(* PLC project ammonium-nitrates, Generated TextualNotationConverter 1.0 *)
(* stored: creationDateTime 2025-07-30T12:00:00, modificationDateTime 2025-09-27T11:37:37 *)

FUNCTION_BLOCK ANALOG_IN
  VAR_INPUT
    Name : STRING;
    Description : STRING;
    Raw_Signal : REAL;
    PV_High : REAL;
    PV_Low : REAL;
    Scaling_Slope : REAL;
    Scaling_Offset : REAL;
    Alarm_Enable : BOOL;
  END_VAR
  VAR_OUTPUT
    PV : REAL;
    High_Alarm : BOOL;
    Low_Alarm : BOOL;
    General_Fault : BOOL;
  END_VAR

            
          
END_FUNCTION_BLOCK

FUNCTION_BLOCK BOOL_IN
  VAR_INPUT
    Name : STRING;
    Description : STRING;
    Bool_In : BOOL;
    Alarm_OnTrue : BOOL;
    Alarm_OnFalse : BOOL;
    Latch_Enable : BOOL;
    Reset_Latch : BOOL;
  END_VAR
  VAR_OUTPUT
    Bool_Out : BOOL;
    Alarm_Active : BOOL;
    Latched_Status : BOOL;
  END_VAR

            
          
END_FUNCTION_BLOCK

FUNCTION_BLOCK PID_BASIC
  VAR_INPUT
    Name : STRING;
    Description : STRING;
    AUTO : BOOL;
    PV : REAL;
    SP : REAL;
    MV_MIN : REAL;
    MV_MAX : REAL;
    X0 : REAL;
    KP : REAL;
    TR : REAL;
    TD : REAL;
    PV_High : REAL;
    PV_Low : REAL;
    Deviation_Limit : REAL;
    Inhibit : BOOL;
  END_VAR
  VAR_OUTPUT
    PV_High_Alarm : BOOL;
    PV_Low_Alarm : BOOL;
    Deviation_Alarm : BOOL;
    XOUT : REAL;
  END_VAR

            
          
END_FUNCTION_BLOCK

FUNCTION_BLOCK RATIO_CONTROL
  VAR_INPUT
    Name : STRING;
    Description : STRING;
    Auto : BOOL;
    PrimaryPV : REAL;
    SecondaryPV : REAL;
    RatioSP : REAL;
    Bias : REAL;
    TrimKp : REAL;
    TrimTi : STRING;
    MV_MIN : REAL;
    MV_MAX : REAL;
    ManOut : REAL;
    Inhibit : BOOL;
  END_VAR
  VAR_OUTPUT
    SlaveSP : REAL;
    ActiveRatio : REAL;
    RatioErr : REAL;
  END_VAR

            
          
END_FUNCTION_BLOCK

FUNCTION_BLOCK VALVE_ELECTRIC
  VAR_INPUT
    Name : STRING;
    Description : STRING;
    Control_Signal : REAL;
    Manual_Mode : BOOL;
    Manual_Position : REAL;
    Open_Limit : REAL;
    Close_Limit : REAL;
    Timeout : STRING;
    Inhibit : BOOL;
  END_VAR
  VAR_OUTPUT
    Valve_Position : REAL;
    Feedback_Pos : REAL;
    Valve_Moving : BOOL;
    Position_Error : BOOL;
    Alarm : BOOL;
  END_VAR

            
          
END_FUNCTION_BLOCK

PROGRAM Section2
  VAR
    FIC102_AcidFlow_SP_FromRatio : REAL;
    FT101_AmmoniaFlow_PV : REAL;
    LT104_ReactorLevel_PV : REAL;
    PH105_ReactorPH_PV : REAL;
    VS107_Scrubber_Permissive : BOOL;
    VS107_Scrubber_Running_DI : BOOL;
    FT101_Raw_mA : REAL;
    FT102_Raw_mA : REAL;
    LT104_Raw_mA : REAL;
    PH105_Raw_mA : REAL;
    TIC103_Temperature_PV : REAL;
  END_VAR
  VAR
    FFIC-102 : RATIO_CONTROL;
    FIC-102 : PID_BASIC;
    FIC-101 : PID_BASIC;
    TIC-103 : PID_BASIC;
    FT-101 : ANALOG_IN;
    FT-102 : ANALOG_IN;
    LT-104 : ANALOG_IN;
    PH-105 : ANALOG_IN;
    FV-102 : VALVE_ELECTRIC;
    FV-101 : VALVE_ELECTRIC;
    VS-107 : BOOL_IN;
  END_VAR
  VAR  (* added by the conversion: wires and edge detectors of the diagram *)
    _OR1_OUT : BOOL;
    _OR3_OUT : BOOL;
  END_VAR

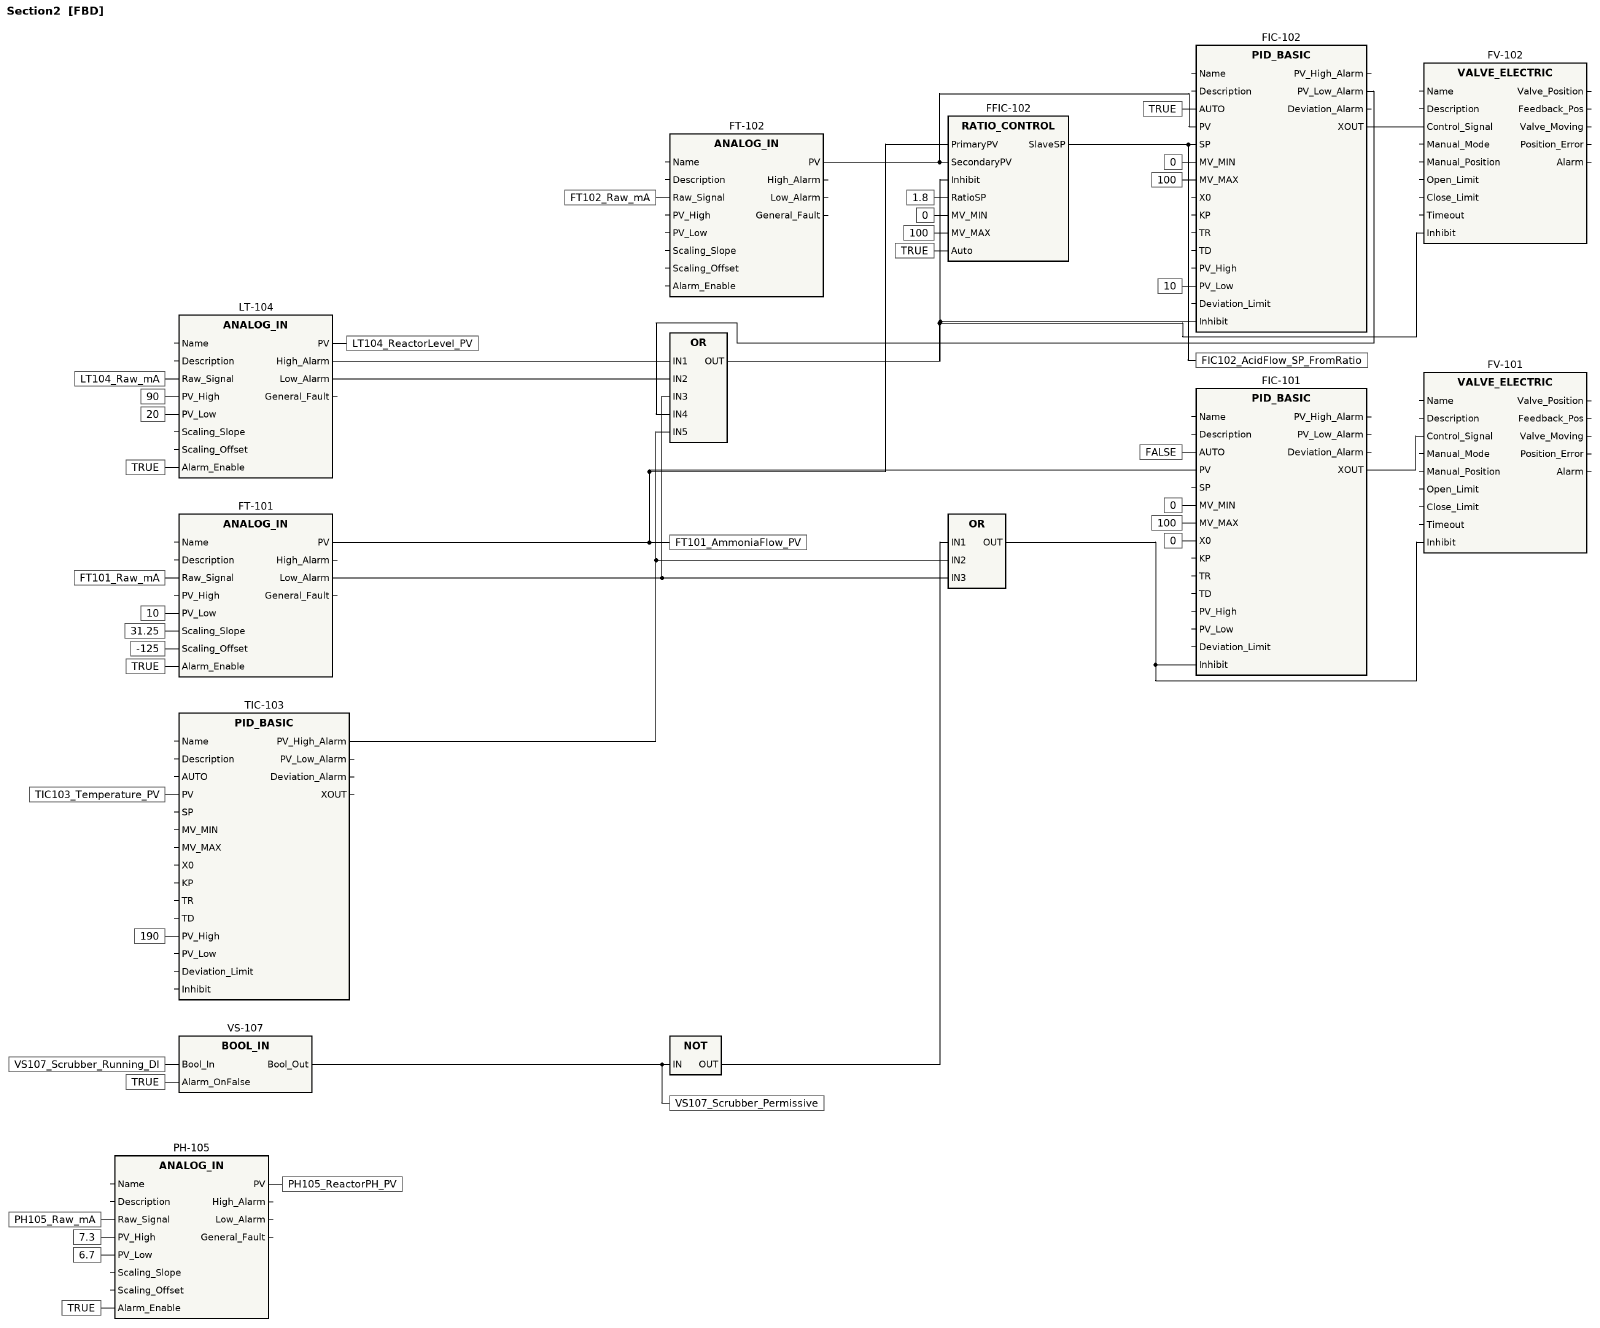
(* FBD diagram, written out as Structured Text *)
FT-101(Raw_Signal := FT101_Raw_mA, PV_Low := 10, Scaling_Slope := 31.25, Scaling_Offset := -125, Alarm_Enable := TRUE);
FT-102(Raw_Signal := FT102_Raw_mA);
LT-104(Raw_Signal := LT104_Raw_mA, PV_High := 90, PV_Low := 20, Alarm_Enable := TRUE);
FIC-102(AUTO := TRUE, PV := FT-102.PV, SP := FFIC-102.SlaveSP, MV_MIN := 0, MV_MAX := 100, PV_Low := 10, Inhibit := _OR1_OUT);
TIC-103(PV := TIC103_Temperature_PV, PV_High := 190);
_OR1_OUT := LT-104.High_Alarm OR LT-104.Low_Alarm OR FT-101.Low_Alarm OR FIC-102.PV_Low_Alarm OR TIC-103.PV_High_Alarm;
FFIC-102(PrimaryPV := FT-101.PV, SecondaryPV := FT-102.PV, Inhibit := _OR1_OUT, RatioSP := 1.8, MV_MIN := 0, MV_MAX := 100, Auto := TRUE);
FIC102_AcidFlow_SP_FromRatio := FFIC-102.SlaveSP;
FT101_AmmoniaFlow_PV := FT-101.PV;
LT104_ReactorLevel_PV := LT-104.PV;
PH-105(Raw_Signal := PH105_Raw_mA, PV_High := 7.3, PV_Low := 6.7, Alarm_Enable := TRUE);
PH105_ReactorPH_PV := PH-105.PV;
VS-107(Bool_In := VS107_Scrubber_Running_DI, Alarm_OnFalse := TRUE);
VS107_Scrubber_Permissive := VS-107.Bool_Out;
_OR3_OUT := NOT VS-107.Bool_Out OR TIC-103.PV_High_Alarm OR FT-101.Low_Alarm;
FIC-101(AUTO := FALSE, PV := FT-101.PV, MV_MIN := 0, MV_MAX := 100, X0 := 0, Inhibit := _OR3_OUT);
FV-102(Control_Signal := FIC-102.XOUT, Inhibit := _OR1_OUT);
FV-101(Control_Signal := FIC-101.XOUT, Inhibit := _OR3_OUT);
END_PROGRAM

FUNCTION_BLOCK DIGITAL_IN
  VAR_INPUT
    Name : STRING;
    Description : STRING;
    DI_Raw : BOOL;
    DebounceTime : STRING;
    EnableAlarm : BOOL;
  END_VAR
  VAR_OUTPUT
    DI_Out : BOOL;
    Fault_State : BOOL;
  END_VAR

            
          
END_FUNCTION_BLOCK

FUNCTION_BLOCK DUTY_STANDBY
  VAR_INPUT
    Name : STRING;
    Description : STRING;
    Enable : BOOL;
    StartRequest : BOOL;
    AlternateEnable : BOOL;
    ForcePumpA : BOOL;
    ForcePumpB : BOOL;
    DutyElapsed : BOOL;
    MinRunElapsed : BOOL;
    SwitchoverDelayElapsed : BOOL;
    StartTimeoutElapsed : BOOL;
    PumpA_RunFB : BOOL;
    PumpB_RunFB : BOOL;
    PumpA_Fault : BOOL;
    PumpB_Fault : BOOL;
    Reset : BOOL;
    Inhibit : BOOL;
  END_VAR
  VAR_OUTPUT
    CmdPumpA : BOOL;
    CmdPumpB : BOOL;
    ActiveIsA : BOOL;
    SwitchedDueToDuty : BOOL;
    SwitchedDueToFailure : BOOL;
    Alarm_FailedStart_A : BOOL;
    Alarm_FailedStart_B : BOOL;
    Alarm_NoAvailablePump : BOOL;
  END_VAR

            
          
END_FUNCTION_BLOCK

FUNCTION_BLOCK MOTOR_2SPD
  VAR_INPUT
    Name : STRING;
    Description : STRING;
    Start_Cmd : BOOL;
    Stop_Cmd : BOOL;
    Speed_High_Cmd : BOOL;
    Speed_Low_Cmd : BOOL;
    Inhibit : BOOL;
  END_VAR
  VAR_OUTPUT
    Motor_Start_Out : BOOL;
    FB_Running : BOOL;
    FB_Trip : BOOL;
    FB_HighSpeed : BOOL;
    FB_LowSpeed : BOOL;
    Alarm_Speed_Error : BOOL;
  END_VAR

            
          
END_FUNCTION_BLOCK

FUNCTION_BLOCK MOTOR_ON_OFF
  VAR_INPUT
    Name : STRING;
    Description : STRING;
    Start_Cmd : BOOL;
    Stop_Cmd : BOOL;
    Start_Delay : STRING;
    MinRunTime : STRING;
    Inhibit : BOOL;
  END_VAR
  VAR_OUTPUT
    Motor_Start_Out : BOOL;
    FB_Running : BOOL;
    FB_Trip : BOOL;
    Alarm_Start_Fail : BOOL;
    Alarm_Stop_Fail : BOOL;
  END_VAR

            
          
END_FUNCTION_BLOCK

FUNCTION_BLOCK MOTOR_VSD
  VAR_INPUT
    Name : STRING;
    Description : STRING;
    Start_Cmd : BOOL;
    Stop_Cmd : BOOL;
    Speed_SP : REAL;
    Accel_Ramp : STRING;
    Decel_Ramp : STRING;
    Inhibit : BOOL;
  END_VAR
  VAR_OUTPUT
    Speed_Out : REAL;
    FB_Running : BOOL;
    FB_Fault : BOOL;
    FB_Ready : BOOL;
    FB_ActualSpeed : REAL;
    Alarm_Speed_Deviation : BOOL;
    Alarm_Comm_Fail : BOOL;
  END_VAR

            
          
END_FUNCTION_BLOCK

FUNCTION_BLOCK SPLIT_RANGE
  VAR_INPUT
    Name : STRING;
    Description : STRING;
    IN : REAL;
    Split_Point : REAL;
    Output1_Start : REAL;
    Output1_End : REAL;
    Output2_Start : REAL;
    Output2_End : REAL;
  END_VAR
  VAR_OUTPUT
    OUT1 : REAL;
    OUT2 : REAL;
  END_VAR

            
          
END_FUNCTION_BLOCK

FUNCTION_BLOCK VALVE_ON_OFF
  VAR_INPUT
    Name : STRING;
    Description : STRING;
    Open_Cmd : BOOL;
    Close_Cmd : BOOL;
    Timeout : STRING;
    Inhibit : BOOL;
  END_VAR
  VAR_OUTPUT
    FB_Opened : BOOL;
    FB_Closed : BOOL;
    Valve_Open_Out : BOOL;
    Valve_Close_Out : BOOL;
    Alarm_Position_Error : BOOL;
    Alarm_General : BOOL;
  END_VAR

            
          
END_FUNCTION_BLOCK

FUNCTION_BLOCK VOTING_ANALOG
  VAR_INPUT
    Name : STRING;
    Description : STRING;
    Input1 : REAL;
    Input2 : REAL;
    Input3 : REAL;
    Deviation_Limit : REAL;
    Voting_Scheme : STRING;
    EnableAlarm : BOOL;
    Inhibit : BOOL;
  END_VAR
  VAR_OUTPUT
    Voted_Output : REAL;
    Sensor1_Fault : BOOL;
    Sensor2_Fault : BOOL;
    Sensor3_Fault : BOOL;
    Alarm_Voting_Error : BOOL;
    Healthy_Sensors_Count : INT;
  END_VAR

            
          
END_FUNCTION_BLOCK

PROGRAM Section3
  VAR
    TIC201_RSP_to_FIC102 : REAL;
  END_VAR
  VAR
    TT-103 : ANALOG_IN;
    TT-104 : ANALOG_IN;
    PT-203 : ANALOG_IN;
    TIC-201 : PID_BASIC;
    FIC-102 : PID_BASIC;
    FV-102 : VALVE_ELECTRIC;
    PV-106 : VALVE_ELECTRIC;
    XV-101 : VALVE_ON_OFF;
    P-205 : MOTOR_ON_OFF;
    HS-204 : DIGITAL_IN;
    VS-206 : DIGITAL_IN;
  END_VAR
  VAR  (* added by the conversion: wires and edge detectors of the diagram *)
    _OR281_OUT : BOOL;
    _OR282_OUT : BOOL;
    _OR283_OUT : BOOL;
  END_VAR

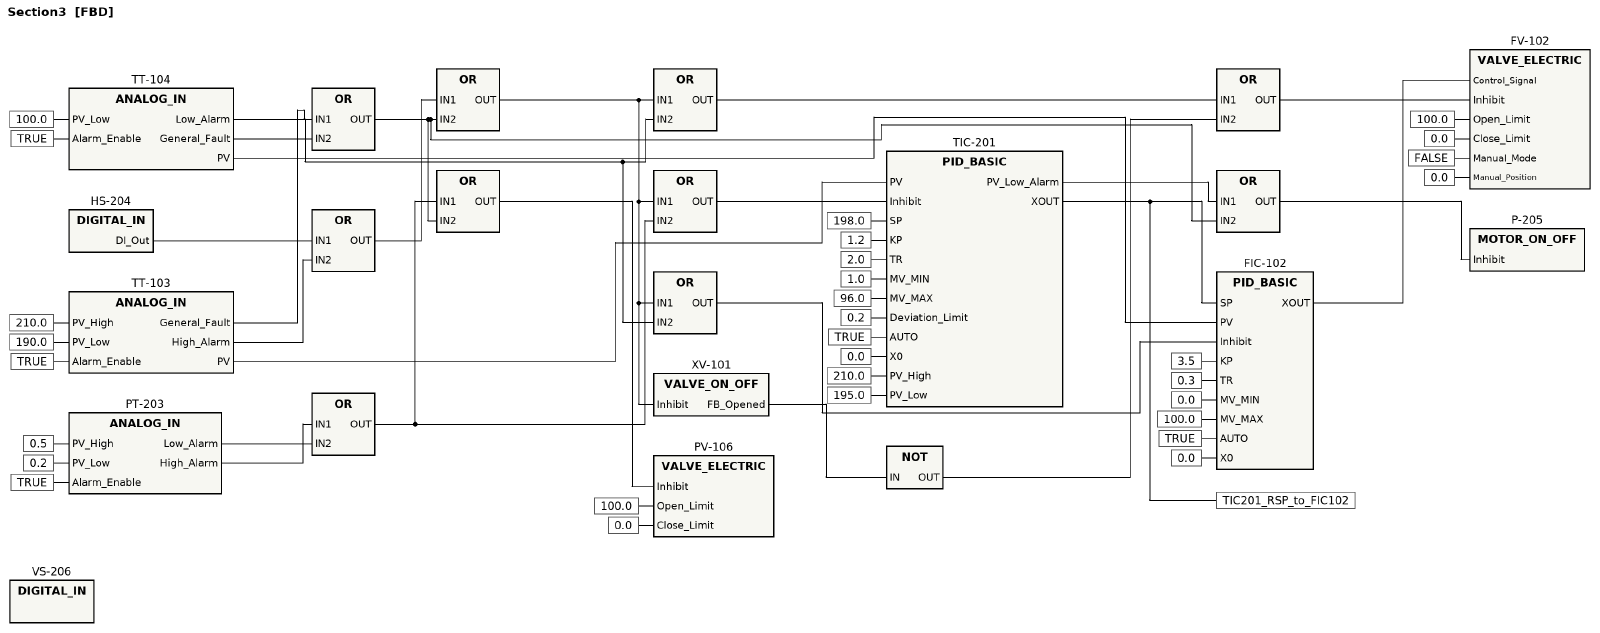
(* FBD diagram, written out as Structured Text *)
TT-103(PV_High := 210.0, PV_Low := 190.0, Alarm_Enable := TRUE);
HS-204();
TT-104(PV_Low := 100.0, Alarm_Enable := TRUE);
_OR281_OUT := TT-103.General_Fault OR TT-104.General_Fault;
_OR282_OUT := HS-204.DI_Out OR TT-103.High_Alarm OR _OR281_OUT;
PT-203(PV_High := 0.5, PV_Low := 0.2, Alarm_Enable := TRUE);
_OR283_OUT := PT-203.High_Alarm OR PT-203.Low_Alarm;
TIC-201(PV := TT-103.PV, Inhibit := _OR282_OUT OR _OR283_OUT, SP := 198.0, KP := 1.2, TR := 2.0, MV_MIN := 1.0, MV_MAX := 96.0, Deviation_Limit := 0.2, AUTO := TRUE, X0 := 0.0, PV_High := 210.0, PV_Low := 195.0);
TIC201_RSP_to_FIC102 := TIC-201.XOUT;
XV-101(Inhibit := _OR282_OUT);
FIC-102(SP := TIC-201.XOUT, PV := TT-104.PV, Inhibit := _OR282_OUT OR TT-104.Low_Alarm, KP := 3.5, TR := 0.3, MV_MIN := 0.0, MV_MAX := 100.0, AUTO := TRUE, X0 := 0.0);
FV-102(Control_Signal := FIC-102.XOUT, Inhibit := _OR282_OUT OR TT-104.Low_Alarm OR NOT XV-101.FB_Opened, Open_Limit := 100.0, Close_Limit := 0.0, Manual_Mode := FALSE, Manual_Position := 0.0);
PV-106(Inhibit := _OR283_OUT OR _OR281_OUT, Open_Limit := 100.0, Close_Limit := 0.0);
P-205(Inhibit := TIC-201.PV_Low_Alarm OR _OR281_OUT);
VS-206();
END_PROGRAM

PROGRAM Section4
  VAR
    RTD302_BedTemp_PV : REAL;
    FT301_Flow_PV : REAL;
    TIC302_RSP_to_FIC301 : REAL;
    FIC301_MV_Out_to_FV301 : REAL;
    AT303_Humidity_PV : REAL;
    PR305_TowerPressure_PV : REAL;
    VS304_Vibration_PV : REAL;
  END_VAR
  VAR
    AT-303 : ANALOG_IN;
    FIC-301 : PID_BASIC;
    FT-301 : ANALOG_IN;
    FV-301 : VALVE_ELECTRIC;
    PR-305 : ANALOG_IN;
    RTD-302 : ANALOG_IN;
    TIC-302 : PID_BASIC;
    VS-304 : ANALOG_IN;
    GR-306 : BOOL_IN;
  END_VAR

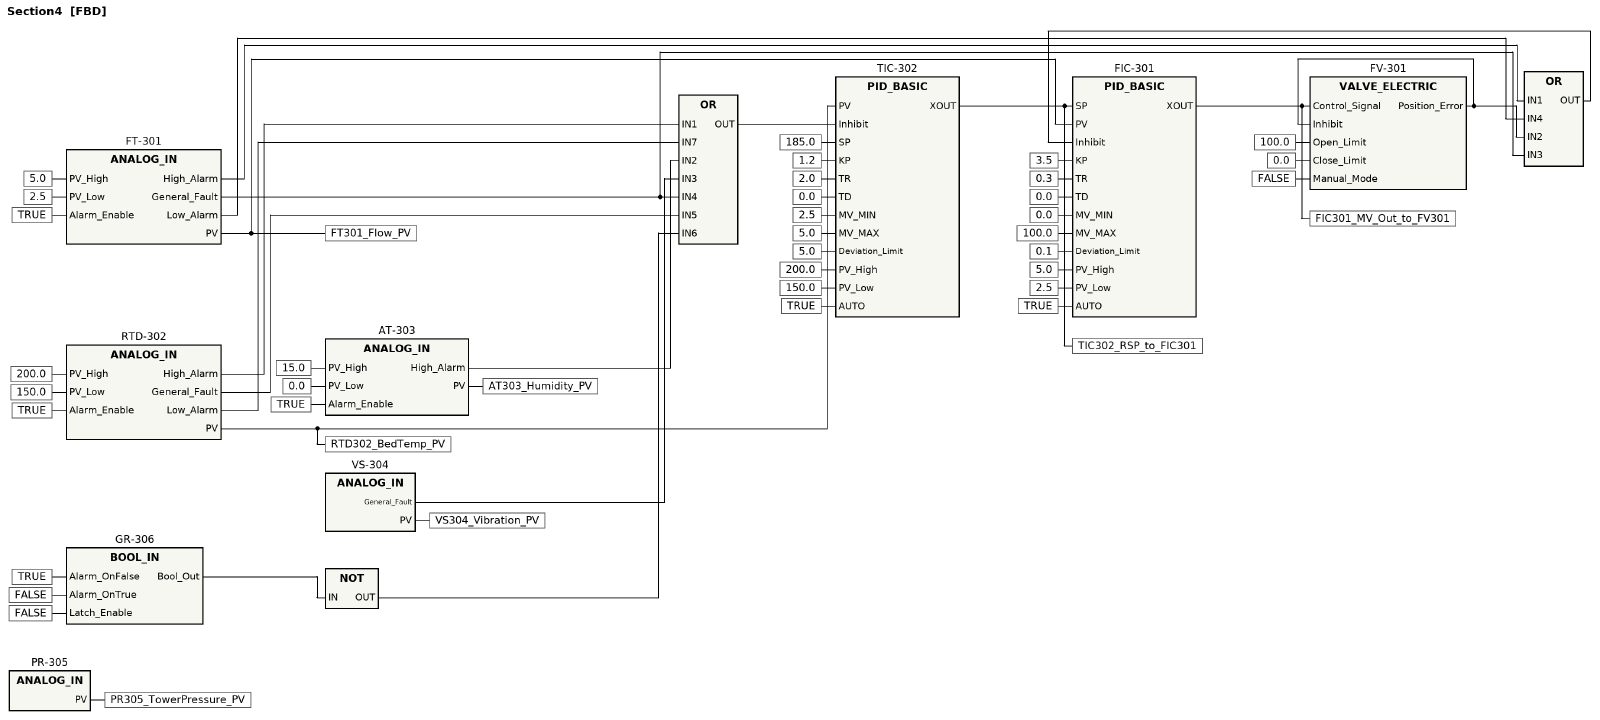
(* FBD diagram, written out as Structured Text *)
AT-303(PV_High := 15.0, PV_Low := 0.0, Alarm_Enable := TRUE);
AT303_Humidity_PV := AT-303.PV;
RTD-302(PV_High := 200.0, PV_Low := 150.0, Alarm_Enable := TRUE);
VS-304();
FT-301(PV_High := 5.0, PV_Low := 2.5, Alarm_Enable := TRUE);
GR-306(Alarm_OnFalse := TRUE, Alarm_OnTrue := FALSE, Latch_Enable := FALSE);
TIC-302(PV := RTD-302.PV, Inhibit := RTD-302.High_Alarm OR RTD-302.Low_Alarm OR AT-303.High_Alarm OR VS-304.General_Fault OR FT-301.General_Fault OR RTD-302.General_Fault OR NOT GR-306.Bool_Out, SP := 185.0, KP := 1.2, TR := 2.0, TD := 0.0, MV_MIN := 2.5, MV_MAX := 5.0, Deviation_Limit := 5.0, PV_High := 200.0, PV_Low := 150.0, AUTO := TRUE);
FV-301(Control_Signal := FIC-301.XOUT, Inhibit := FV-301.Position_Error, Open_Limit := 100.0, Close_Limit := 0.0, Manual_Mode := FALSE);
FIC-301(SP := TIC-302.XOUT, PV := FT-301.PV, Inhibit := FT-301.High_Alarm OR FT-301.Low_Alarm OR FV-301.Position_Error OR FT-301.General_Fault, KP := 3.5, TR := 0.3, TD := 0.0, MV_MIN := 0.0, MV_MAX := 100.0, Deviation_Limit := 0.1, PV_High := 5.0, PV_Low := 2.5, AUTO := TRUE);
FIC301_MV_Out_to_FV301 := FIC-301.XOUT;
FT301_Flow_PV := FT-301.PV;
PR-305();
PR305_TowerPressure_PV := PR-305.PV;
RTD302_BedTemp_PV := RTD-302.PV;
TIC302_RSP_to_FIC301 := TIC-302.XOUT;
VS304_Vibration_PV := VS-304.PV;
END_PROGRAM

PROGRAM Section5
  VAR
    TT401_CoolerOutletTemp_PV : REAL;
    FT402_AntiCakingFlow_PV : REAL;
    TIC401_RSP_to_FIC402 : REAL;
    FIC402_MV_to_FV402 : REAL;
    FIC402_SP_Manual : REAL;
  END_VAR
  VAR
    TIC-401 : PID_BASIC;
    TT-401 : ANALOG_IN;
    FIC-402 : PID_BASIC;
    FT-402 : ANALOG_IN;
    FV-402 : VALVE_ELECTRIC;
    MP-405 : MOTOR_ON_OFF;
    PS-403 : BOOL_IN;
    PSA-404 : DIGITAL_IN;
  END_VAR
  VAR  (* added by the conversion: wires and edge detectors of the diagram *)
    _OR184_OUT : BOOL;
  END_VAR

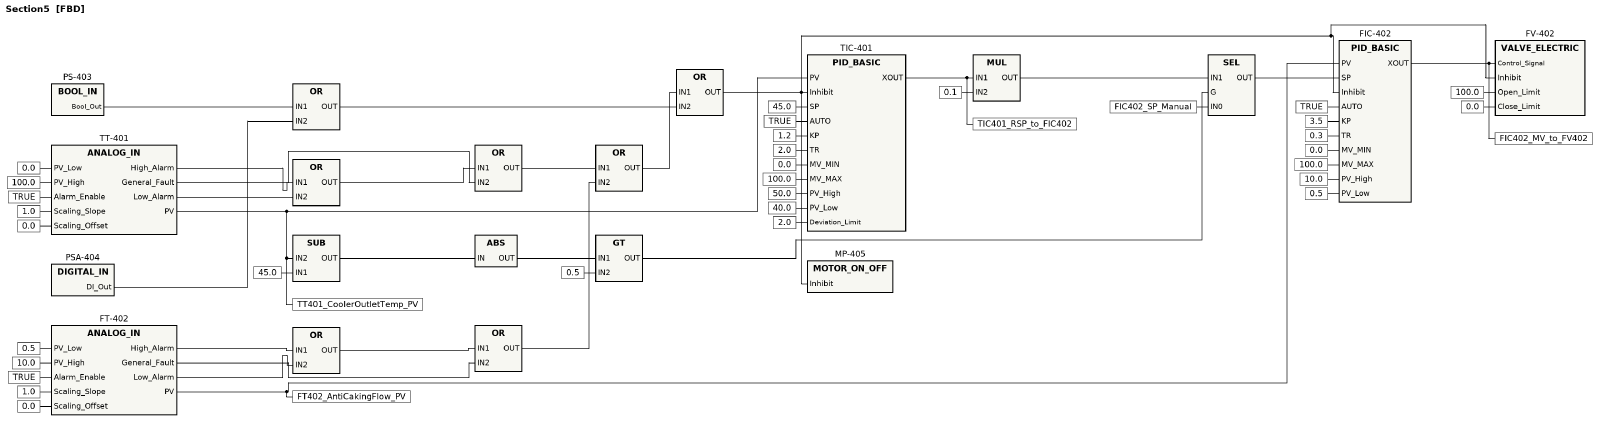
(* FBD diagram, written out as Structured Text *)
FT-402(PV_Low := 0.5, PV_High := 10.0, Alarm_Enable := TRUE, Scaling_Slope := 1.0, Scaling_Offset := 0.0);
TT-401(PV_Low := 0.0, PV_High := 100.0, Alarm_Enable := TRUE, Scaling_Slope := 1.0, Scaling_Offset := 0.0);
PS-403();
PSA-404();
_OR184_OUT := TT-401.High_Alarm OR TT-401.Low_Alarm OR TT-401.General_Fault OR FT-402.High_Alarm OR FT-402.Low_Alarm OR FT-402.General_Fault OR PS-403.Bool_Out OR PSA-404.DI_Out;
TIC-401(PV := TT-401.PV, Inhibit := _OR184_OUT, SP := 45.0, AUTO := TRUE, KP := 1.2, TR := 2.0, MV_MIN := 0.0, MV_MAX := 100.0, PV_High := 50.0, PV_Low := 40.0, Deviation_Limit := 2.0);
FIC-402(PV := FT-402.PV, SP := SEL(TIC-401.XOUT * 0.1, ABS(TT-401.PV - 45.0) > 0.5, FIC402_SP_Manual), Inhibit := _OR184_OUT, AUTO := TRUE, KP := 3.5, TR := 0.3, MV_MIN := 0.0, MV_MAX := 100.0, PV_High := 10.0, PV_Low := 0.5);
FIC402_MV_to_FV402 := FIC-402.XOUT;
FT402_AntiCakingFlow_PV := FT-402.PV;
TIC401_RSP_to_FIC402 := TIC-401.XOUT;
TT401_CoolerOutletTemp_PV := TT-401.PV;
FV-402(Control_Signal := FIC-402.XOUT, Inhibit := _OR184_OUT, Open_Limit := 100.0, Close_Limit := 0.0);
MP-405(Inhibit := _OR184_OUT);
END_PROGRAM

PROGRAM Section6
  VAR
    LT501_Level_Pct : REAL;
    WB505_Flow_Pct : REAL;
    RIC506_SC504_FlowSP : REAL;
    Ratio_Bias_Manual : REAL;
  END_VAR
  VAR
    LT-501 : ANALOG_IN;
    WB-505 : ANALOG_IN;
    AP-503 : VALVE_ON_OFF;
    PRV-502 : VALVE_ON_OFF;
    RIC-506 : RATIO_CONTROL;
    FIC-507 : PID_BASIC;
    SC-504 : MOTOR_VSD;
  END_VAR
  VAR  (* added by the conversion: wires and edge detectors of the diagram *)
    _OR232_OUT : BOOL;
    _GT233_OUT : BOOL;
    _LT234_OUT : BOOL;
  END_VAR

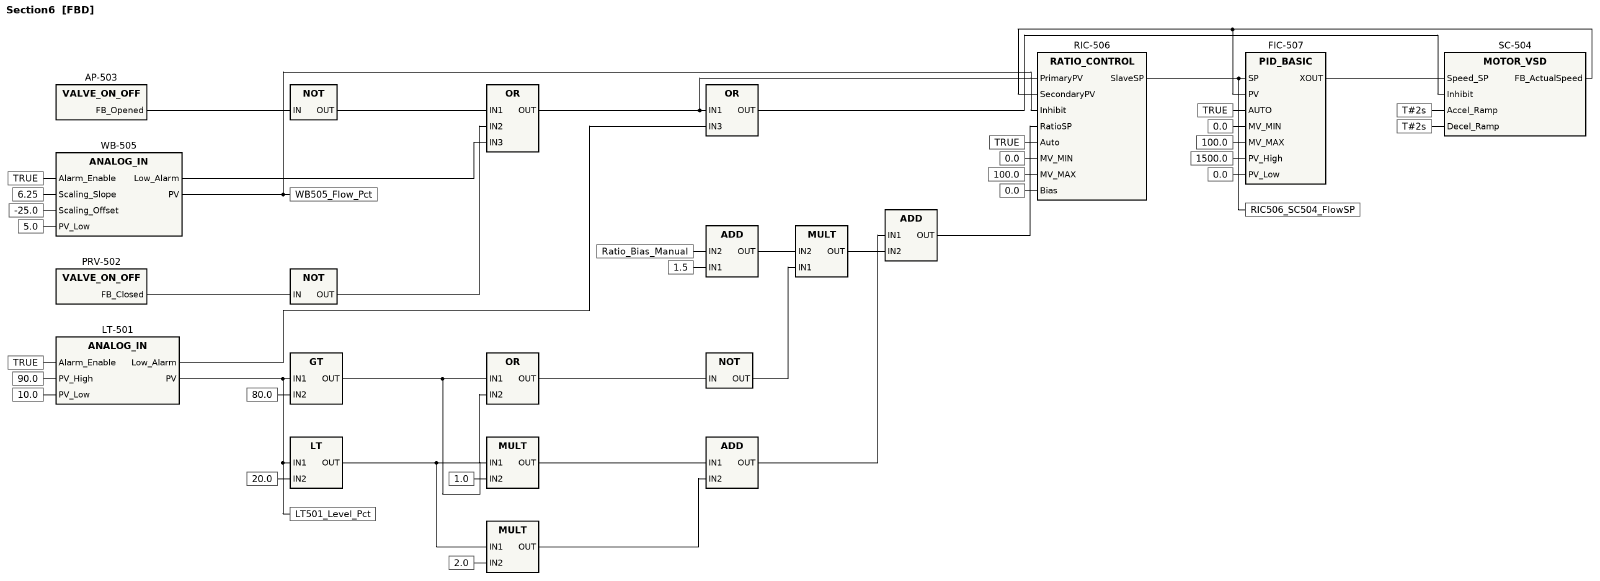
(* FBD diagram, written out as Structured Text *)
LT-501(Alarm_Enable := TRUE, PV_High := 90.0, PV_Low := 10.0);
LT501_Level_Pct := LT-501.PV;
WB-505(Alarm_Enable := TRUE, Scaling_Slope := 6.25, Scaling_Offset := -25.0, PV_Low := 5.0);
FIC-507(SP := RIC-506.SlaveSP, PV := SC-504.FB_ActualSpeed, AUTO := TRUE, MV_MIN := 0.0, MV_MAX := 100.0, PV_High := 1500.0, PV_Low := 0.0);
AP-503();
PRV-502();
_OR232_OUT := NOT AP-503.FB_Opened OR NOT PRV-502.FB_Closed OR WB-505.Low_Alarm;
SC-504(Speed_SP := FIC-507.XOUT, Inhibit := _OR232_OUT OR LT-501.Low_Alarm, Accel_Ramp := T#2s, Decel_Ramp := T#2s);
_GT233_OUT := LT-501.PV > 80.0;
_LT234_OUT := LT-501.PV < 20.0;
RIC-506(PrimaryPV := WB-505.PV, SecondaryPV := SC-504.FB_ActualSpeed, Inhibit := _OR232_OUT, RatioSP := MULT(_GT233_OUT, 1.0) + MULT(_LT234_OUT, 2.0) + MULT(Ratio_Bias_Manual + 1.5, NOT (_GT233_OUT OR _LT234_OUT)), Auto := TRUE, MV_MIN := 0.0, MV_MAX := 100.0, Bias := 0.0);
RIC506_SC504_FlowSP := RIC-506.SlaveSP;
WB505_Flow_Pct := WB-505.PV;
END_PROGRAM

CONFIGURATION Config0
  RESOURCE Res0 ON PLC
    TASK task0(INTERVAL := T#20ms, PRIORITY := 0);
    PROGRAM instance0 WITH task0 : Section2;
    PROGRAM instance_1 WITH task0 : Section3;
    PROGRAM instance_2 WITH task0 : Section4;
    PROGRAM instance_3 WITH task0 : Section5;
    PROGRAM instance_4 WITH task0 : Section6;
  END_RESOURCE
END_CONFIGURATION
